// TIA Portal V20 export
// export: Created 2026-04-11T06:02:30.146765Z, ExportSetting WithDefaults, DisplayName Totally Integrated Automation Portal, DisplayVersion V20, DisplayName TIA Portal Openness, DisplayVersion V20, DisplayName TIA Portal Version Control Interface, DisplayVersion V20, DisplayName STEP 7 Professional, DisplayVersion V20, DisplayName STEP 7 Safety, DisplayVersion V20, DisplayName WinCC Basic/Comfort/Advanced, DisplayVersion V20, DisplayName WinCC Unified, DisplayVersion V20
TYPE "udtError_Sterlco"
// stored: IsFailsafeCompliant false
   STRUCT
      Alarm1State { ExternalWritable := 'False'} : Bool;   // Alarm 1 state
      Alarm2State { ExternalWritable := 'False'} : Bool;   // Alarm 2 state
      Alarm3State { ExternalWritable := 'False'} : Bool;   // Alarm 3 state
      Alarm4State { ExternalWritable := 'False'} : Bool;   // Alarm 4 state
      NotInManual { ExternalWritable := 'False'} : Bool;   // Not in auto mode
      SensorBreak { ExternalWritable := 'False'} : Bool;   // Sensor broken
      LoopBreak { ExternalWritable := 'False'} : Bool;   // Loop broken (open loop)
      HeaterFail { ExternalWritable := 'False'} : Bool;   // Load fault detected
      PV_OutOfRange { ExternalWritable := 'False'} : Bool;   // PV out of table range
      DC_ControlModuleFault { ExternalWritable := 'False'} : Bool;   // DC control module fault
      RemoteInputSensorBreak { ExternalWritable := 'False'} : Bool;   // Remote input sensor broken
      IP1_Fault { ExternalWritable := 'False'} : Bool;   // IP1 Fault
   END_STRUCT;
END_TYPE
